// TIA Portal project "num" (V16)

(* hardware
DEVICE "S71500/ET200MP station_1"  S7-1500 station
   slot 0: "导轨_0"  Rack  6ES7 590-1***0-0AA0
   slot 1: "PLC_1"  CPU 1511-1 PN  6ES7 511-1AK02-0AB0  V2.8
      slot 3: "CPU 显示_1"  6ES7591-1AA00-0AA0
      slot 32768: "PROFINET 接口_1"  X1
         slot 32769: "端口_1"  X1 P1
         slot 32770: "端口_2"  X1 P2
      slot 34817: "Virtual CP interface port_1"  Virtual CP interface port  Virtual CP interface port
*)

// ===== PLC "PLC_1"  CPU 1511-1 PN =====

DATA_BLOCK "数据块_1"   // DB1
{ S7_Optimized_Access := 'FALSE' }
VERSION : 0.1
   VAR
      number : Int;
      number_1 : Real;
      number_3 : Real;
   END_VAR
BEGIN
END_DATA_BLOCK

FUNCTION "块_1" : Void   // FC1, LAD
{ S7_Optimized_Access := 'TRUE' }
VERSION : 0.1
   VAR_INPUT
      IN1 : Int;
      IN2 : Int;
      IN3 : Real;
   END_VAR
   VAR_OUTPUT
      out : Real;
   END_VAR
   VAR_TEMP
      temp1 : Int;
      temp2 : Int;
      temp3 : Real;
      temp4 : Real;
      temp5 : Real;
      temp6 : Real;
      temp7 : Real;
   END_VAR
BEGIN

REGION Network 1
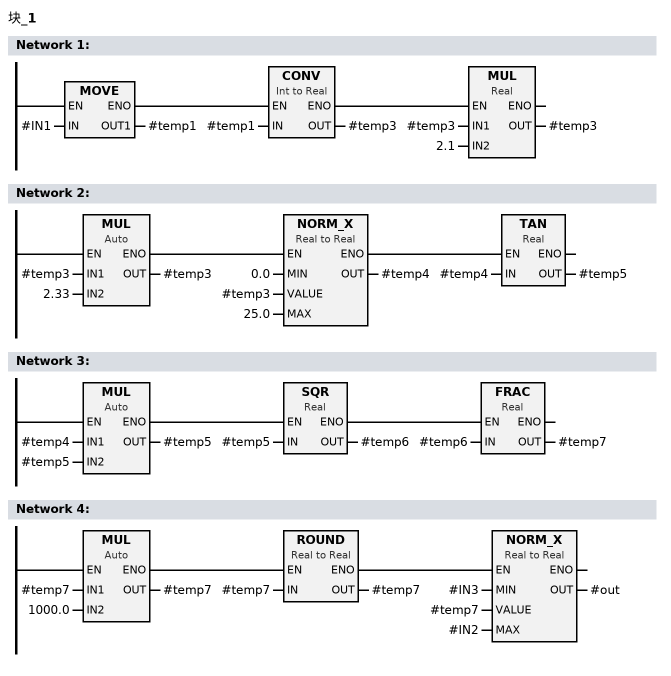
   RUNG wire#powerrail
      Move(in := #IN1, out1 => #temp1)
      { S7_Templates := "[SrcType := Int, DestType := Real]" } Convert(in := #temp1, out => #temp3)
      { S7_Templates := "SrcType := Real" } Mul(in1 := #temp3, in2 := 2.1, out => #temp3)
   END_RUNG
   // the same network as SCL:
   #temp1 := #IN1;
   #temp3 := INT_TO_REAL(#temp1);
   #temp3 := #temp3 * 2.1;
END_REGION

REGION Network 2
   #temp3 := #temp3 * 2.33;
   #temp4 := NORM_X(MIN := 0.0, VALUE := #temp3, MAX := 25.0);
   #temp5 := TAN(#temp4);
END_REGION

REGION Network 3
   #temp5 := #temp4 * #temp5;
   #temp6 := SQR(#temp5);
   #temp7 := FRAC(#temp6);
END_REGION

REGION Network 4
   RUNG wire#powerrail
      Mul(in1 := #temp7, in2 := 1000.0, out => #temp7)
      { S7_Templates := "[SrcType := Real, DestType := Real]" } Round(in := #temp7, out => #temp7)
      { S7_Templates := "[SrcType := Real, DestType := Real]" } Normalize(min := #IN3, value := #temp7, max := #IN2, out => #out)
   END_RUNG
   // the same network as SCL:
   #temp7 := #temp7 * 1000.0;
   #temp7 := ROUND(#temp7);
   #out := NORM_X(MIN := #IN3, VALUE := #temp7, MAX := #IN2);
END_REGION
END_FUNCTION

ORGANIZATION_BLOCK "Main"   // OB1, LAD, ProgramCycle
TITLE = "Main Program Sweep (Cycle)"
{ S7_Optimized_Access := 'TRUE' }
VERSION : 0.1
   VAR_INPUT
      Initial_Call : Bool;   // Initial call of this OB
      Remanence : Bool;   // =True, if remanent data are available
   END_VAR
BEGIN

REGION Network 1
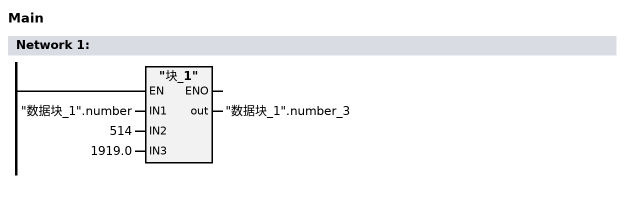
   RUNG wire#powerrail
      "块_1"(IN1 := "数据块_1".number, IN2 := 514, IN3 := 1919.0, out => "数据块_1".number_3)
   END_RUNG
   // the same network as SCL:
   "块_1"(IN1 := "数据块_1".number, IN2 := 514, IN3 := 1919.0, out => "数据块_1".number_3);
END_REGION
END_ORGANIZATION_BLOCK